# EPICS SNL sequencer program: viocs/bo_ps/bo_psApp/src/ps_sp_init.stt
program ps_sp_init

int event_proc;
assign event_proc to "EVENT-BOPS-SP-INIT.PROC";

ss ss1 {
    state init {
        when (delay(2.0)) {
            event_proc = 1;
            pvPut(event_proc);
        } exit
    }
}
